TYPE DUT_stMarkingData :
STRUCT
    LayoutName 		: STRING(50);
    OrderReference 	: STRING(50);
    ProfileLaser 	: STRING(50);
END_STRUCT
END_TYPE

(* stored: Version 1.1.0.1, ProductVersion 3.1.4024.15
   DUT DUT_stMarkingData: Id {3c16cbc0-9d0a-4fdf-8dd3-54ec000d859f} *)
